PROGRAM MAIN
VAR
	myStateMachine : StateMachine();
END_VAR

// Call Program
myStateMachine();

END_PROGRAM

(* stored: Version 1.1.0.1, ProductVersion 3.1.4024.12
   POU MAIN: Id {b8ddf703-70a7-4ad2-8e3e-66f68b5d2cba}, SpecialFunc None *)
